// TwinCAT 3 PLC project PLC1
// ProgramVersion: 3.1.4024.0
// libraries:
//   Tc2_Standard, * (Beckhoff Automation GmbH)
//   Tc2_System, * (Beckhoff Automation GmbH)
//   Tc3_Module, * (Beckhoff Automation GmbH)
// project tree:
//   DUTs/ EL3443_FullDUT.TcDUT, EL3443_Phase_Basic.TcDUT, EL3443_Phase_Power.TcDUT, EL3443_Phase_Status.TcDUT
//   / PlcTask.TcTTO
//   POUs/ MAIN.TcPOU
// real-time tasks:
//   TASK PlcTask: cycle T#10ms, priority 20, ADS port 350
// I/O:
//   DEVICE Device 1 (EtherCAT) (disabled), AmsNetId 10.199.163.130.2.1
//     Term 1 (EK1100) [EK1100 EtherCAT Coupler (2A E-Bus)]
//       Term 2 (EL3443) [EL3443 3Ch. Power Measuring]

CONFIGURATION PLC1
    RESOURCE PLC ON TwinCAT3
        TASK PlcTask(INTERVAL := T#10ms, PRIORITY := 20);
        PROGRAM MAIN WITH PlcTask : MAIN;
    END_RESOURCE
END_CONFIGURATION

// ---- DUTs/EL3443_FullDUT.TcDUT
TYPE EL3443_FullDUT :
STRUCT
END_STRUCT
END_TYPE

// ---- DUTs/EL3443_Phase_Basic.TcDUT
TYPE EL3443_Phase_Basic :
STRUCT
END_STRUCT
END_TYPE

// ---- DUTs/EL3443_Phase_Power.TcDUT
TYPE EL3443_Phase_Power :
STRUCT
END_STRUCT
END_TYPE

// ---- DUTs/EL3443_Phase_Status.TcDUT
TYPE EL3443_Phase_Status :
STRUCT
END_STRUCT
END_TYPE

// ---- POUs/MAIN.TcPOU
PROGRAM MAIN
VAR
END_VAR

(* Application Engineer: LucasK *)
(* MQTT Sample to TecnoProcess Test *) 
(* Using Mosquitto MQTT Open Source Server *)
(* And MQTT-Explorer to test *)
(* start mosquitto with net start mosquitto *)

END_PROGRAM
